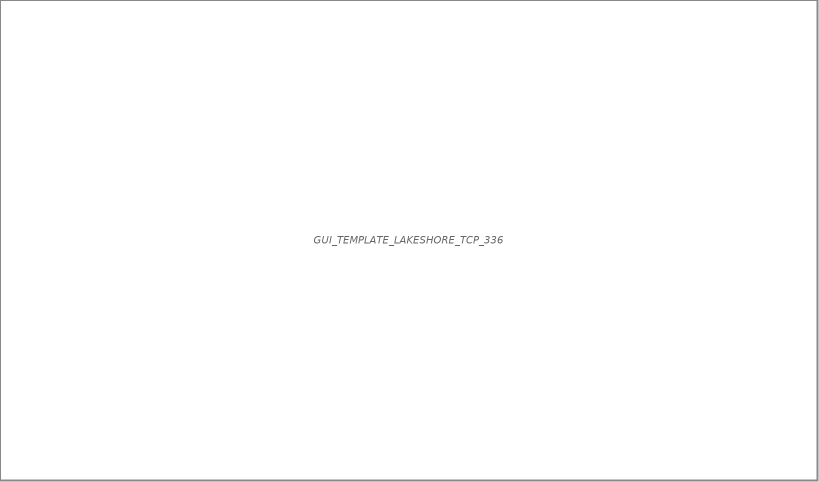
VISUALIZATION GUI_LAKESHORE_TCP_336  // 819x482
    Frame (0,0 817x480)
        shows GUI_TEMPLATE_LAKESHORE_TCP_336(m_Instance := MAIN.LS336_TCP)
END_VISUALIZATION

(* stored: Version 1.1.0.1, ProductVersion 3.1.4022.16
   Visu GUI_LAKESHORE_TCP_336: Id {9c04f4f8-a0fb-485d-bd8b-c64090302dfc} *)
